PROGRAM ElevationControl
VAR_INPUT
	// enable the axis
	enable: 	BOOL;
	// reset an error
	reset:		BOOL;
	// increase the eleveation
	up:			BOOL;
	// decrease the elevation
	down:		BOOL;
	// set position of the axis in degrees
	position:	LREAL;
	// set the Velocity of the axis
	velocity:	LREAL;
	// move axis command
	MoveAxis:	BOOL;
	// calibrate the axis
	HomeAxis:	BOOL;
	// enable tracking
	Tracking:	BOOL;
	// stop the Axis
	StopAxis:	BOOL;
	// reset diagnostic errors
	bSoEReset:	 	BOOL;
END_VAR
VAR_OUTPUT
	// axis is ready to operate
	Ready:			BOOL;
	// drive error condition
	error: 			BOOL;
	// warning condition
	warning:		BOOL;
	// actual position of the elevation axis
	actual_position: 	LREAL;
	// error ID of the elevation axis
	ErrorID: 		UDINT;
	// axis is calibrated
	Calibrated:		BOOL;
	// time to reach target position
	slewtime:		LREAL;
END_VAR
VAR
	ElevationAxis:			FB_Axis2;
	ElevationCalibration: 	MC_SetPosition;
	fbSoEReset: 			FB_SoEReset;
	// delay until commutator angle is measured
	readydelay:				TON;
	// disable trigger for hydraulics
	enable_trigger:			F_TRIG;
	// store last position
	getlastposition:		BOOL := TRUE;
	ElevationAxisEvent: 	FB_Eventlog;
	ElevationDiagnosticEvent: 	FB_Eventlog;
	ElevationBrakeEvent: 	FB_Eventlog;
	HighElevationEvent: 	FB_Eventlog;
	LowElevationEvent:		FB_Eventlog;
	TorqueWarning:			FB_EventLog;
	CalibrationEvent:		FB_Eventlog;
	// elevation torque in percent
	elevation_torque: 		REAL;
	// timer to trigger a warning if torque is high
	torque_timer:			TON;
	ReadParameter:			MC_ReadParameter;
	DiagnosticError:		BOOL;
END_VAR
VAR CONSTANT
	// current position of the calibration cam. Apply an offset here if necessary
	calibration_position:	LREAL := 30.55; //30.4; //45.399; // offset = +1.26 from 44.139; //44.061; //43.806122; //42.1281; //43.000
END_VAR
VAR PERSISTENT
	last_position:	LREAL := -1.0;
END_VAR

// limit the position input to a sane value
position := LIMIT(0.0, position, 90.0);

IF Calibrated AND (actual_position > 89.0 OR actual_position < 1.0) THEN
	Tracking := FALSE;
END_IF

//if we enable the axis, we have to open the brake first
IF Enable THEN
	IF NOT Calibrated THEN
		CoverControl.open := TRUE;
		IF CoverControl.isopen THEN
			HydraulicsControl.open_brake();
		END_IF
	ELSE
		HydraulicsControl.open_brake();
	END_IF
	
END_IF

enable_trigger(CLK := enable);
// close the brake on the falling edge of the enable signal
IF enable_trigger.Q THEN
	HydraulicsControl.close_brake();
END_IF

IF ElevationAxis.Calibrated OR Error THEN
	HomeAxis := FALSE;
END_IF

Calibrated := ElevationAxis.Calibrated;

IF HomeAxis THEN
	position := calibration_position;
	MoveAxis := FALSE;
	Tracking := FALSE;
END_IF

IF MoveAxis OR StopAxis THEN
	Tracking := FALSE;
END_IF

// if NOT Enabled and ActVelo>1 then issue a warning
warning := NOT enable AND GVL_Telescope.ElevationAxisRef.NcToPlc.ActVelo>2.0;

// deactivate limit switches on homing
MC_SetAcceptBlockedDriveSignal(
	Axis := GVL_Telescope.ElevationAxisRef, 
	Enable := HomeAxis);
	
ElevationAxis(
	Enable := 			enable AND HydraulicsControl.brake_open,
	Reset := 			reset,
	MoveAxis :=			MoveAxis,
	HomeAxis :=			HomeAxis,
	StopAxis :=			StopAxis,
	Tracking :=			Tracking,
	Position := 		position, 
	Velocity :=			Velocity,
	Enable_Positive :=  GVL_Telescope.Elevation_inputs.0 OR HomeAxis,
	Enable_Negative := 	GVL_Telescope.Elevation_inputs.1,
	Jog_Forward :=		up,
	Jog_Backwards := 	down,
	bCalibrationCam :=	NOT GVL_Telescope.Elevation_inputs.0,
	ActualPosition => 	actual_position,
	Error => 			error,
	ErrorID => 			ErrorID,
	AxisRef :=			GVL_Telescope.ElevationAxisRef);

IF ElevationAxis.MoveDone THEN
	MoveAxis := FALSE;
END_IF

IF ElevationAxis.HomeDone THEN
	HomeAxis := FALSE;
END_IF
	
IF ElevationAxis.ResetDone THEN
	reset := FALSE;
END_IF

IF ElevationAxis.StopDone THEN
	StopAxis := FALSE;
END_IF

DiagnosticError := FALSE;
IF GVL_Telescope.Elevation_diagnostic < 16#D012 AND GVL_Telescope.Elevation_diagnostic > 16#D014 THEN
	DiagnosticError :=TRUE;
	ErrorID := GVL_Telescope.Elevation_diagnostic;
END_IF

ElevationCalibration(Axis := GVL_Telescope.ElevationAxisRef,
	Execute := getlastposition AND last_position>=0.0 AND NOT Calibrated,
	Position := last_position);

IF ElevationCalibration.Done THEN
	getlastposition := FALSE;
END_IF

IF Calibrated THEN
	last_position := actual_position;
END_IF

IF bSoEReset THEN
	last_position := -1.0;
	fbSoEReset(
		Axis := GVL_Telescope.ElevationAxisRef,
		Execute := TRUE,
		Timeout := DEFAULT_ADS_TIMEOUT);
 	IF NOT fbSoEReset.Busy THEN
		fbSoEReset(Axis := GVL_Telescope.ElevationAxisRef, Execute := FALSE);
		bSoEReset := FALSE;
		Reset := TRUE;
	END_IF
END_IF 

readydelay(IN :=  HydraulicsControl.brake_open, PT := T#6000MS, Q=> ready);

ReadParameter(	Axis := GVL_Telescope.ElevationAxisRef, 
				Enable := ElevationAxis.InMotion, 
				ParameterNumber := MC_AxisParameter.AxisRemainingTimeToGo, 
				ReadMode := E_ReadMode.READMODE_CYCLIC);
				
IF ReadParameter.Valid THEN
	slewtime := ReadParameter.Value;
END_IF

elevation_torque := GVL_Telescope.Elevation_torque / 10.0;
torque_timer(IN := ABS(elevation_torque) > 50.0, PT := T#1000MS);
		
ElevationAxisEvent(	Trigger := Error, 
				Level := ADSLOG_MSGTYPE_ERROR,
				FormatString := 'Elevation Axis Error: %s',
				OnMessage := NCError_TO_STRING(ErrorID));

ElevationDiagnosticEvent(	
	Trigger := 		DiagnosticError, 
	Level := 		ADSLOG_MSGTYPE_ERROR,
	FormatString :=	'Elevation Axis Diagnostic Error: %s',
	OnMessage := 	NCError_TO_STRING(GVL_Telescope.Elevation_diagnostic));

				
HighElevationEvent(	Trigger := Calibrated AND actual_position > 85.0, 
				Level := ADSLOG_MSGTYPE_WARN,
				FormatString := 'High Elevation: %s',
				OnMessage := LREAL_TO_FMTSTR(actual_position, 2, TRUE));

LowElevationEvent(	Trigger := Calibrated AND actual_position < 5.0, 
				Level := ADSLOG_MSGTYPE_WARN,
				FormatString := 'Low Elevation: %s',
				OnMessage := LREAL_TO_FMTSTR(actual_position, 2, TRUE));
				
ElevationBrakeEvent( Trigger := NOT enable AND HydraulicsControl.brake_open, 
				Level := ADSLOG_MSGTYPE_WARN,
				FormatString := '%s',
				OnMessage := 'Brake was opened without elevation axis enabled!'); 

TorqueWarning(	
	Trigger := torque_timer.Q, 
	Level := 		ADSLOG_MSGTYPE_WARN,
	FormatString :=	'%s',
	OnMessage := 	'Elevation torque is high.');
	
CalibrationEvent(
	Trigger :=	Calibrated,
	Level :=	ADSLOG_MSGTYPE_HINT,
	OnMessage := 'Elevation is calibrated.'
	);

END_PROGRAM

(* stored: Version 1.1.0.1, ProductVersion 3.1.4024.9
   POU ElevationControl: Id {c0371b19-3d1d-4f20-bd19-ce60539d69cd}, SpecialFunc None *)
